// TIA Portal V19 export
ORGANIZATION_BLOCK "Main"   // OB1, LAD, ProgramCycle
TITLE = "Main Program Sweep (Cycle)"
{ S7_Optimized_Access := 'TRUE' }
// stored: SetENOAutomatically false
   VAR_INPUT
      Initial_Call : Bool;   // Initial call of this OB
      Remanence : Bool;   // =True, if remanent data are available
   END_VAR
BEGIN

REGION Network 1
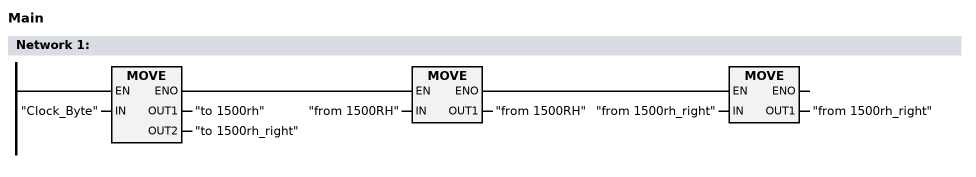
   RUNG wire#powerrail
      Move(in := "Clock_Byte", out1 => "to 1500rh", out2 => "to 1500rh_right")
      Move(in := "from 1500RH", out1 => "from 1500RH")
      Move(in := "from 1500rh_right", out1 => "from 1500rh_right")
   END_RUNG
   // the same network as SCL:
   "to 1500rh" := "Clock_Byte";
   "to 1500rh_right" := "Clock_Byte";
   "from 1500RH" := "from 1500RH";
   "from 1500rh_right" := "from 1500rh_right";
END_REGION
END_ORGANIZATION_BLOCK
